Omron CX-Programmer project NewProject (CX-Programmer 9.75)

# PLC NewPLC1: CJ2M CPU31
I/O table (CPU CJ2M-CPU31): rack 0 slot 0 CJ1W-ID211; rack 0 slot 1 CJ1W-OD212; rack 0 slot 11 CJ2M-EIP21

## Global symbols (name address type ; comment)
1.00 BOOL  ; Motor On
W0.00 BOOL  ; Motor Run
C0000 BOOL  ; If sensor read 5 times
0 CHANNEL  ; Counter
0.00 BOOL  ; Sensor NO
1 CHANNEL  ; Add this
1.01 BOOL  ; Lamp
C0 CHANNEL  ; Reset
D0 CHANNEL  ; New address
D0.00 BOOL  ; Memory Address
T0000 BOOL  ; If motor run for 30 sec
T0001 BOOL  ; Stuck
T0100 BOOL  ; if motor run for 30 sec
W0.01 BOOL  ; Stuck

## Program NewProgram1 (cyclic task 0)
Local symbols
P_0_5s BOOL

### Section Section1

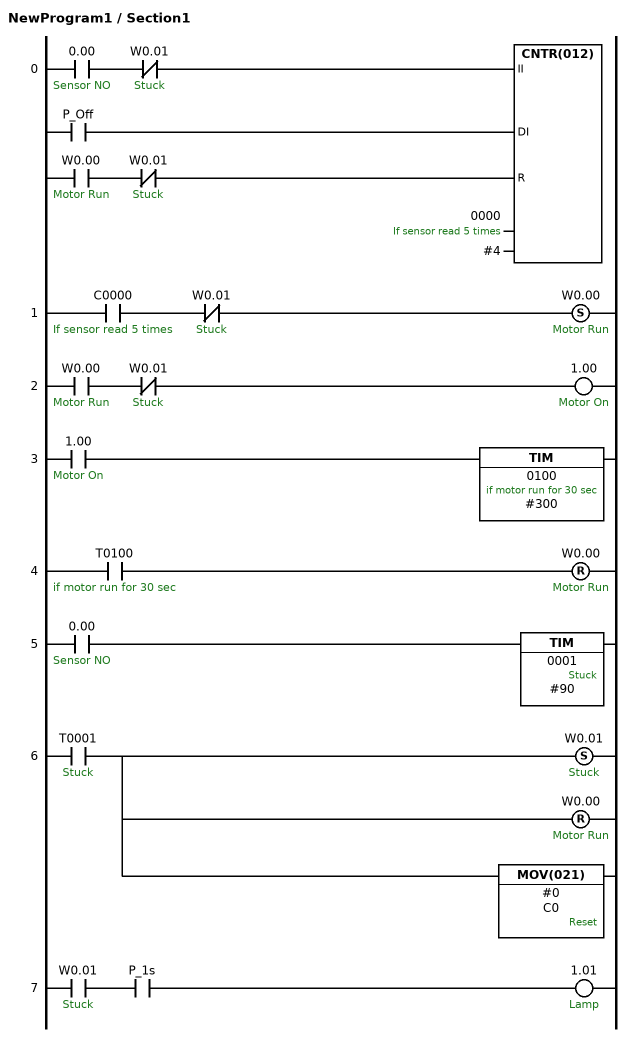
; rung 0
LD 0.00  ; Sensor NO
ANDNOT W0.01  ; Stuck
LD P_Off
LD W0.00  ; Motor Run
ANDNOT W0.01  ; Stuck
CNTR(012) 0000 #4  ; If sensor read 5 times
; rung 1
LD C0000  ; If sensor read 5 times
ANDNOT W0.01  ; Stuck
SET W0.00  ; Motor Run
; rung 2
LD W0.00  ; Motor Run
ANDNOT W0.01  ; Stuck
OUT 1.00  ; Motor On
; rung 3
LD 1.00  ; Motor On
TIM 0100 #300  ; if motor run for 30 sec
; rung 4
LD T0100  ; if motor run for 30 sec
RSET W0.00  ; Motor Run
; rung 5
LD 0.00  ; Sensor NO
TIM 0001 #90  ; Stuck
; rung 6
LD T0001  ; Stuck
SET W0.01  ; Stuck
RSET W0.00  ; Motor Run
MOV(021) #0 C0  ; Reset
; rung 7
LD W0.01  ; Stuck
AND P_1s
OUT 1.01  ; Lamp
; rung 8
END(001)